// Mitsubishi GX Works2 project: exam_prep_diagrams   PLC: Q02/Q02H

PROGRAM complex1
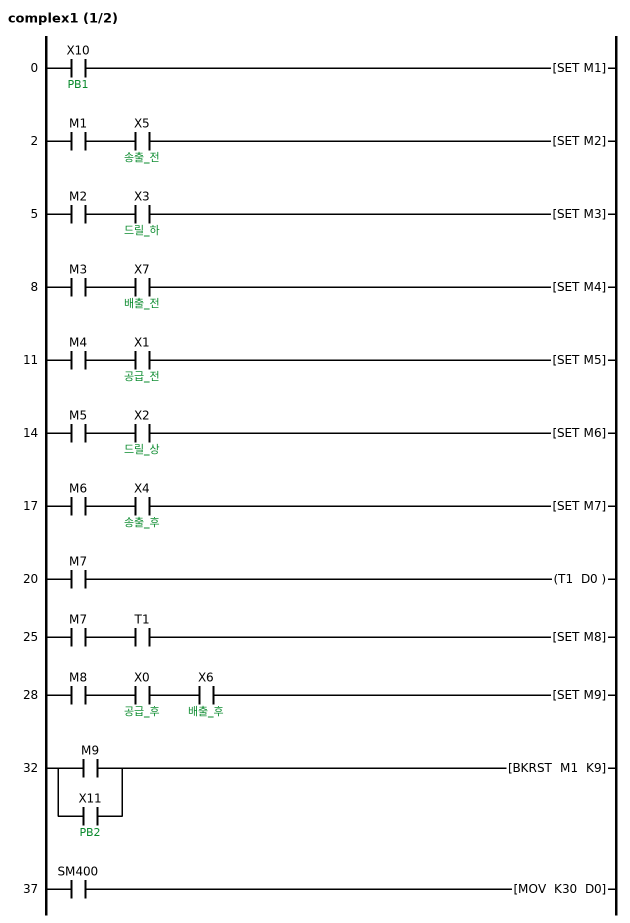
0     LD      X10  ; PB1
      SET     M1
2     LD      M1
      AND     X5  ; 송출_전
      SET     M2
5     LD      M2
      AND     X3  ; 드릴_하
      SET     M3
8     LD      M3
      AND     X7  ; 배출_전
      SET     M4
11    LD      M4
      AND     X1  ; 공급_전
      SET     M5
14    LD      M5
      AND     X2  ; 드릴_상
      SET     M6
17    LD      M6
      AND     X4  ; 송출_후
      SET     M7
20    LD      M7
      OUT     T1 D0
25    LD      M7
      AND     T1
      SET     M8
28    LD      M8
      AND     X0  ; 공급_후
      AND     X6  ; 배출_후
      SET     M9
32    LD      M9
      OR      X11  ; PB2
      BKRST   M1 K9
37    LD      SM400
      MOV     K30 D0
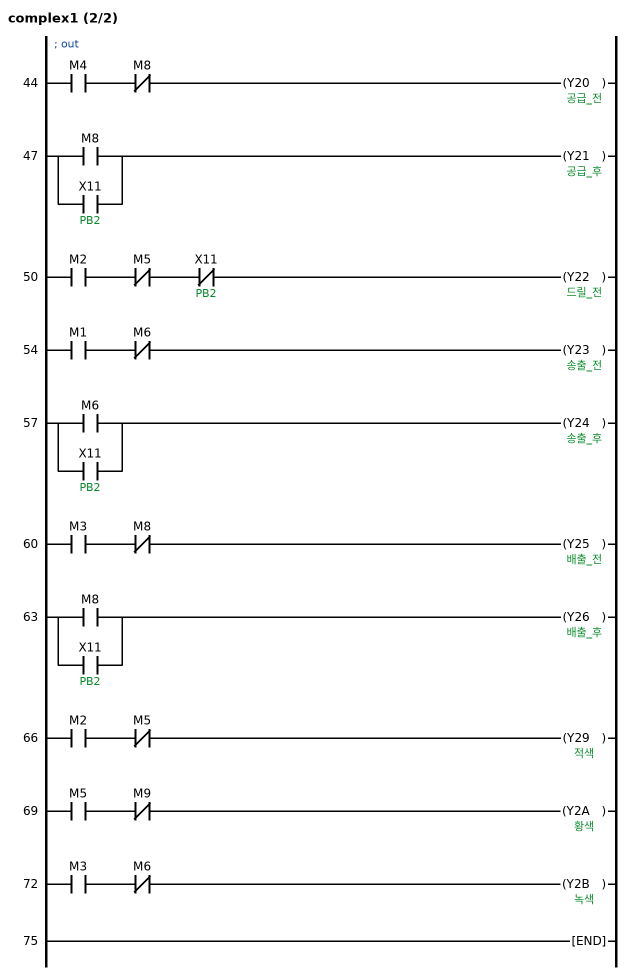
; out
44    LD      M4
      ANI     M8
      OUT     Y20  ; 공급_전
47    LD      M8
      OR      X11  ; PB2
      OUT     Y21  ; 공급_후
50    LD      M2
      ANI     M5
      ANI     X11  ; PB2
      OUT     Y22  ; 드릴_전
54    LD      M1
      ANI     M6
      OUT     Y23  ; 송출_전
57    LD      M6
      OR      X11  ; PB2
      OUT     Y24  ; 송출_후
60    LD      M3
      ANI     M8
      OUT     Y25  ; 배출_전
63    LD      M8
      OR      X11  ; PB2
      OUT     Y26  ; 배출_후
66    LD      M2
      ANI     M5
      OUT     Y29  ; 적색
69    LD      M5
      ANI     M9
      OUT     Y2A  ; 황색
72    LD      M3
      ANI     M6
      OUT     Y2B  ; 녹색
75    END
END_PROGRAM

PROGRAM complex2
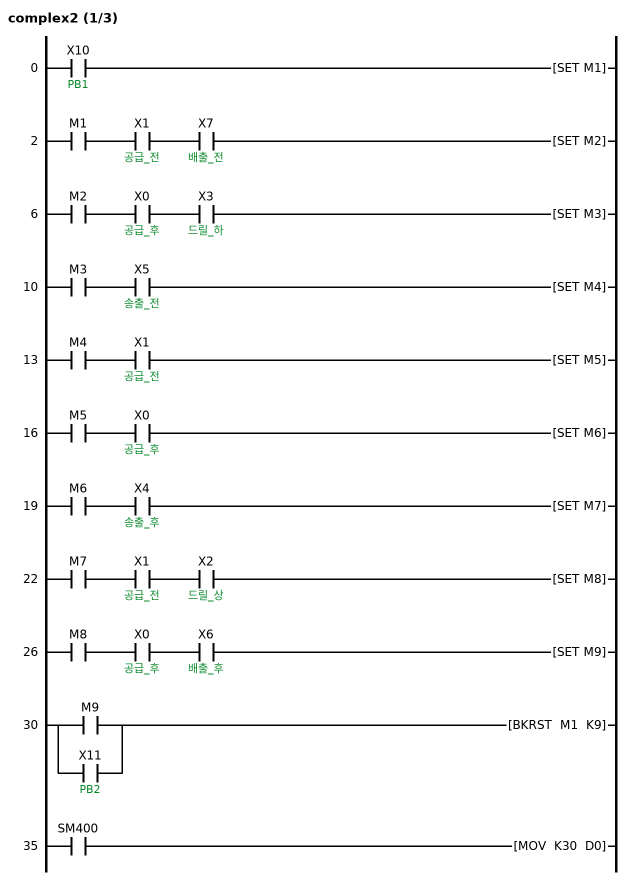
0     LD      X10  ; PB1
      SET     M1
2     LD      M1
      AND     X1  ; 공급_전
      AND     X7  ; 배출_전
      SET     M2
6     LD      M2
      AND     X0  ; 공급_후
      AND     X3  ; 드릴_하
      SET     M3
10    LD      M3
      AND     X5  ; 송출_전
      SET     M4
13    LD      M4
      AND     X1  ; 공급_전
      SET     M5
16    LD      M5
      AND     X0  ; 공급_후
      SET     M6
19    LD      M6
      AND     X4  ; 송출_후
      SET     M7
22    LD      M7
      AND     X1  ; 공급_전
      AND     X2  ; 드릴_상
      SET     M8
26    LD      M8
      AND     X0  ; 공급_후
      AND     X6  ; 배출_후
      SET     M9
30    LD      M9
      OR      X11  ; PB2
      BKRST   M1 K9
35    LD      SM400
      MOV     K30 D0
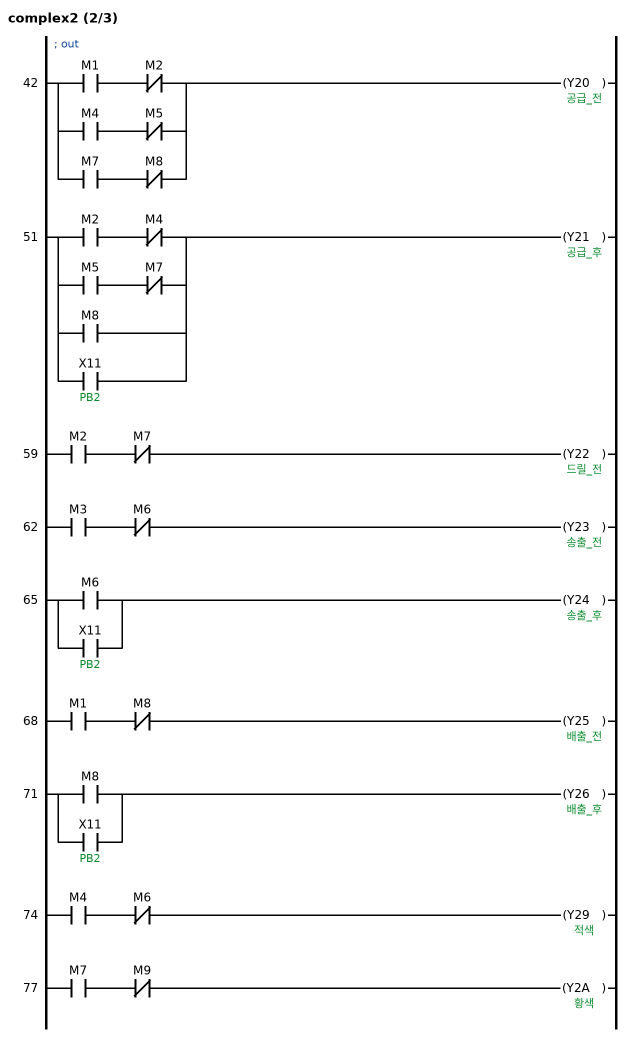
; out
42    LD      M1
      ANI     M2
      LD      M4
      ANI     M5
      ORB
      LD      M7
      ANI     M8
      ORB
      OUT     Y20  ; 공급_전
51    LD      M2
      ANI     M4
      LD      M5
      ANI     M7
      ORB
      OR      M8
      OR      X11  ; PB2
      OUT     Y21  ; 공급_후
59    LD      M2
      ANI     M7
      OUT     Y22  ; 드릴_전
62    LD      M3
      ANI     M6
      OUT     Y23  ; 송출_전
65    LD      M6
      OR      X11  ; PB2
      OUT     Y24  ; 송출_후
68    LD      M1
      ANI     M8
      OUT     Y25  ; 배출_전
71    LD      M8
      OR      X11  ; PB2
      OUT     Y26  ; 배출_후
74    LD      M4
      ANI     M6
      OUT     Y29  ; 적색
77    LD      M7
      ANI     M9
      OUT     Y2A  ; 황색
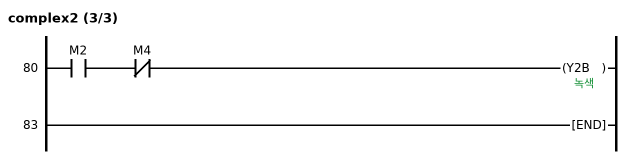
80    LD      M2
      ANI     M4
      OUT     Y2B  ; 녹색
83    END
END_PROGRAM

PROGRAM base
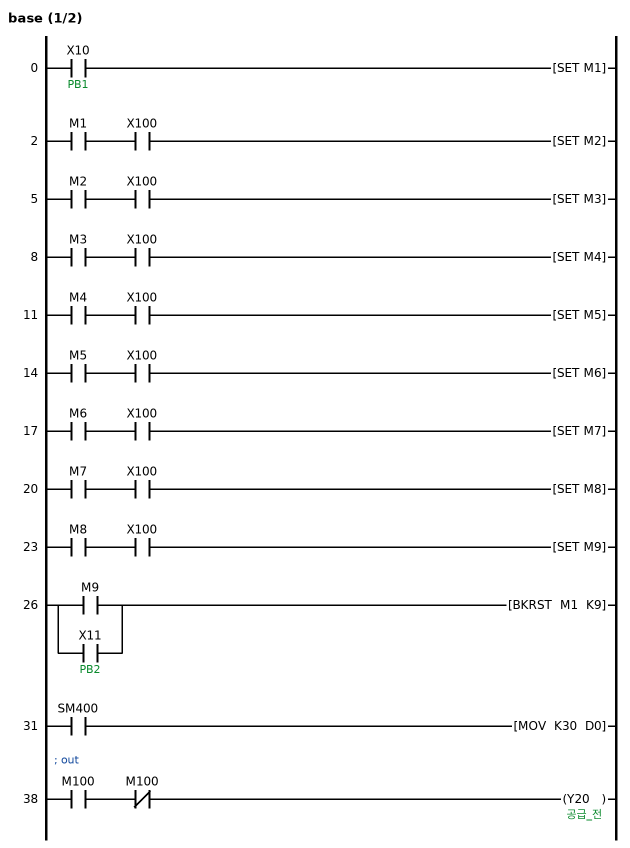
0     LD      X10  ; PB1
      SET     M1
2     LD      M1
      AND     X100
      SET     M2
5     LD      M2
      AND     X100
      SET     M3
8     LD      M3
      AND     X100
      SET     M4
11    LD      M4
      AND     X100
      SET     M5
14    LD      M5
      AND     X100
      SET     M6
17    LD      M6
      AND     X100
      SET     M7
20    LD      M7
      AND     X100
      SET     M8
23    LD      M8
      AND     X100
      SET     M9
26    LD      M9
      OR      X11  ; PB2
      BKRST   M1 K9
31    LD      SM400
      MOV     K30 D0
; out
38    LD      M100
      ANI     M100
      OUT     Y20  ; 공급_전
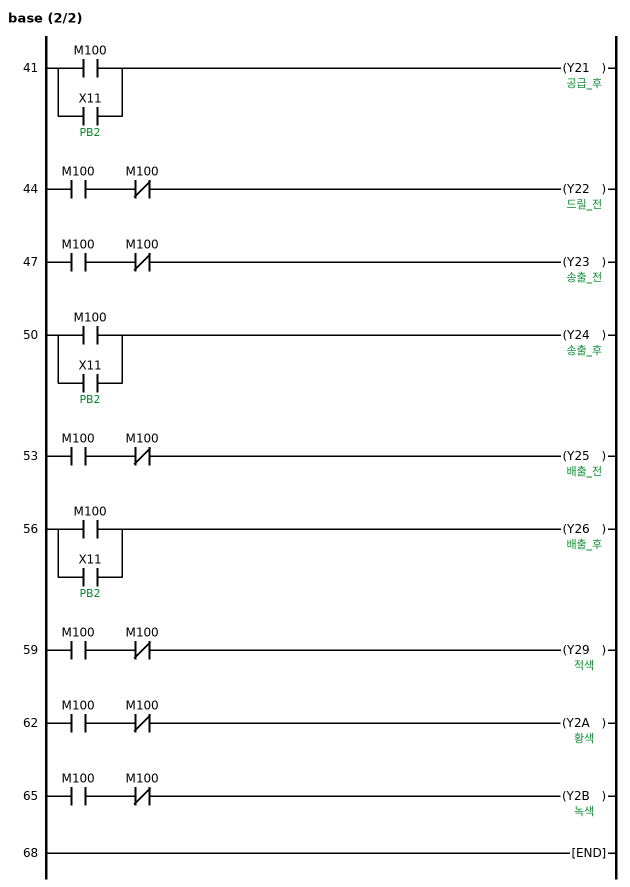
41    LD      M100
      OR      X11  ; PB2
      OUT     Y21  ; 공급_후
44    LD      M100
      ANI     M100
      OUT     Y22  ; 드릴_전
47    LD      M100
      ANI     M100
      OUT     Y23  ; 송출_전
50    LD      M100
      OR      X11  ; PB2
      OUT     Y24  ; 송출_후
53    LD      M100
      ANI     M100
      OUT     Y25  ; 배출_전
56    LD      M100
      OR      X11  ; PB2
      OUT     Y26  ; 배출_후
59    LD      M100
      ANI     M100
      OUT     Y29  ; 적색
62    LD      M100
      ANI     M100
      OUT     Y2A  ; 황색
65    LD      M100
      ANI     M100
      OUT     Y2B  ; 녹색
68    END
END_PROGRAM

PROGRAM complex3
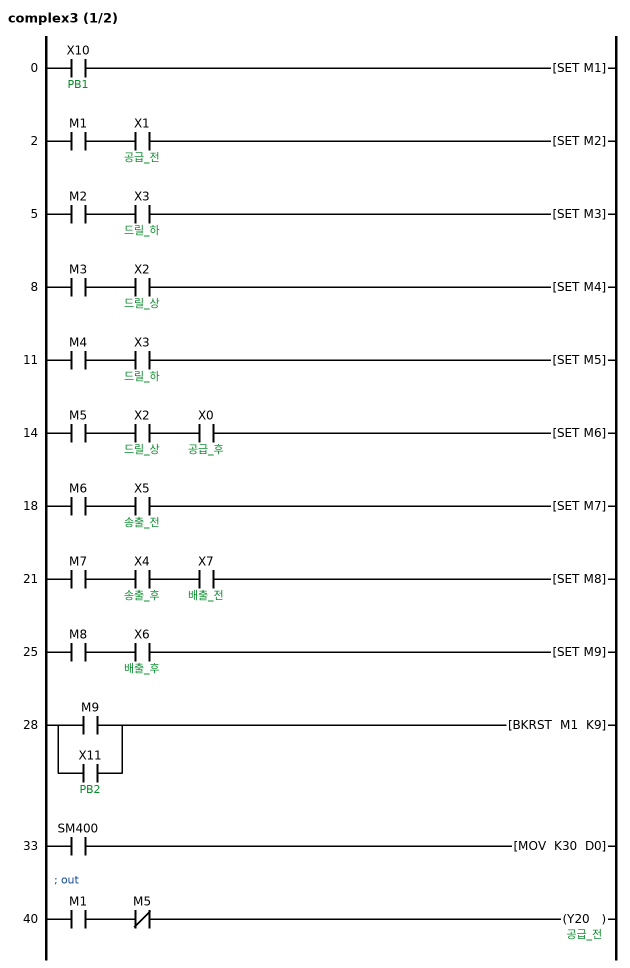
0     LD      X10  ; PB1
      SET     M1
2     LD      M1
      AND     X1  ; 공급_전
      SET     M2
5     LD      M2
      AND     X3  ; 드릴_하
      SET     M3
8     LD      M3
      AND     X2  ; 드릴_상
      SET     M4
11    LD      M4
      AND     X3  ; 드릴_하
      SET     M5
14    LD      M5
      AND     X2  ; 드릴_상
      AND     X0  ; 공급_후
      SET     M6
18    LD      M6
      AND     X5  ; 송출_전
      SET     M7
21    LD      M7
      AND     X4  ; 송출_후
      AND     X7  ; 배출_전
      SET     M8
25    LD      M8
      AND     X6  ; 배출_후
      SET     M9
28    LD      M9
      OR      X11  ; PB2
      BKRST   M1 K9
33    LD      SM400
      MOV     K30 D0
; out
40    LD      M1
      ANI     M5
      OUT     Y20  ; 공급_전
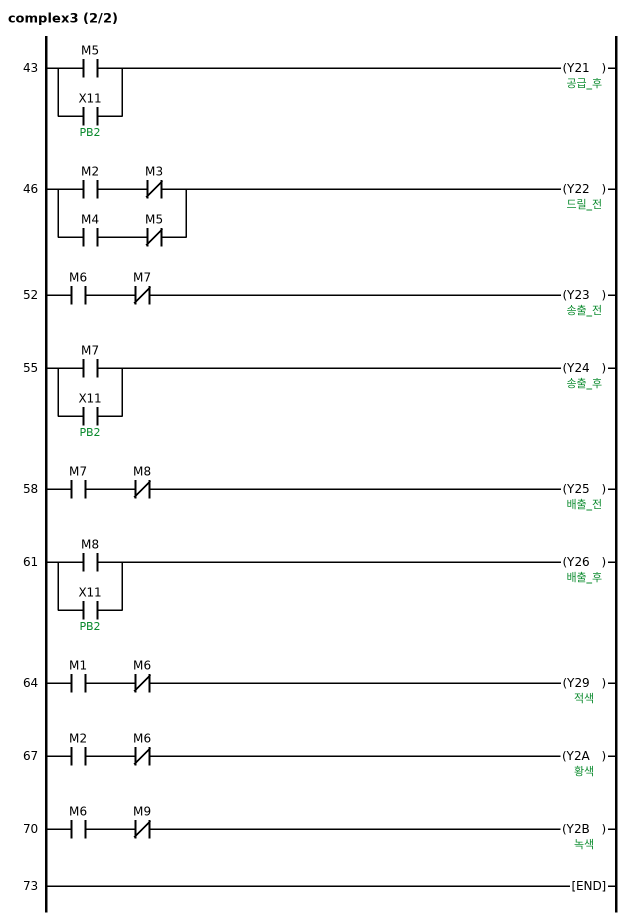
43    LD      M5
      OR      X11  ; PB2
      OUT     Y21  ; 공급_후
46    LD      M2
      ANI     M3
      LD      M4
      ANI     M5
      ORB
      OUT     Y22  ; 드릴_전
52    LD      M6
      ANI     M7
      OUT     Y23  ; 송출_전
55    LD      M7
      OR      X11  ; PB2
      OUT     Y24  ; 송출_후
58    LD      M7
      ANI     M8
      OUT     Y25  ; 배출_전
61    LD      M8
      OR      X11  ; PB2
      OUT     Y26  ; 배출_후
64    LD      M1
      ANI     M6
      OUT     Y29  ; 적색
67    LD      M2
      ANI     M6
      OUT     Y2A  ; 황색
70    LD      M6
      ANI     M9
      OUT     Y2B  ; 녹색
73    END
END_PROGRAM

PROGRAM EXAM1
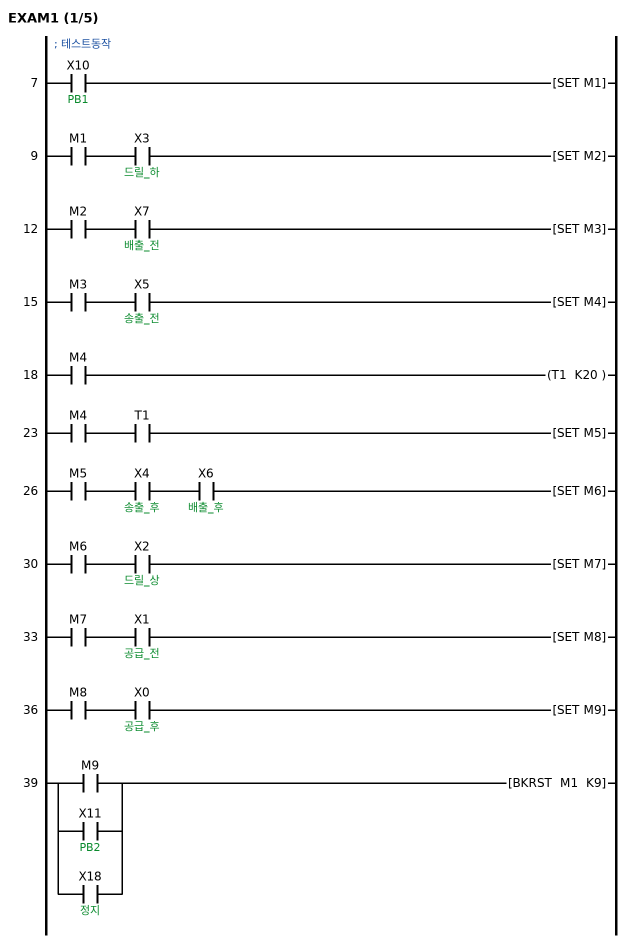
; 테스트동작
7     LD      X10  ; PB1
      SET     M1
9     LD      M1
      AND     X3  ; 드릴_하
      SET     M2
12    LD      M2
      AND     X7  ; 배출_전
      SET     M3
15    LD      M3
      AND     X5  ; 송출_전
      SET     M4
18    LD      M4
      OUT     T1 K20
23    LD      M4
      AND     T1
      SET     M5
26    LD      M5
      AND     X4  ; 송출_후
      AND     X6  ; 배출_후
      SET     M6
30    LD      M6
      AND     X2  ; 드릴_상
      SET     M7
33    LD      M7
      AND     X1  ; 공급_전
      SET     M8
36    LD      M8
      AND     X0  ; 공급_후
      SET     M9
39    LD      M9
      OR      X11  ; PB2
      OR      X18  ; 정지
      BKRST   M1 K9
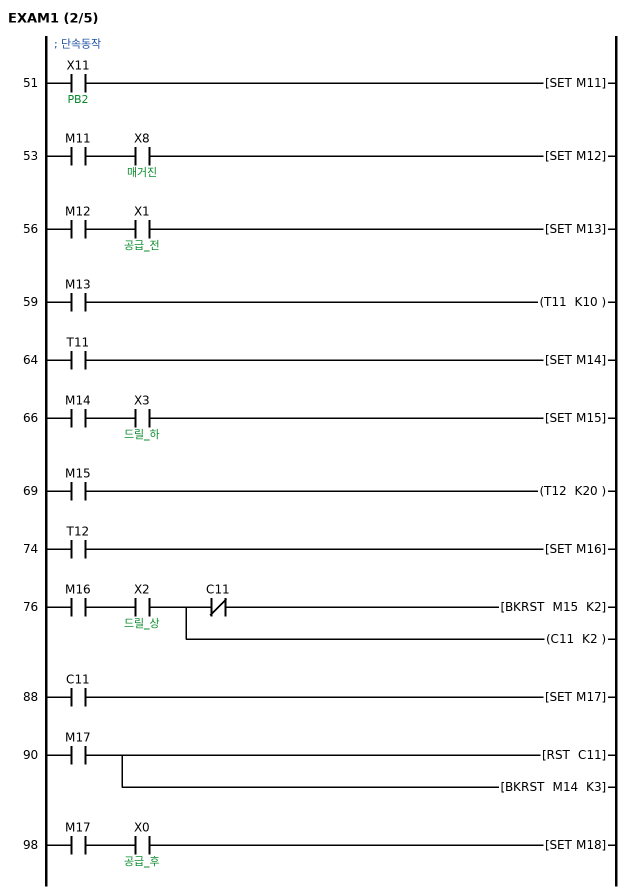
; 단속동작
51    LD      X11  ; PB2
      SET     M11
53    LD      M11
      AND     X8  ; 매거진
      SET     M12
56    LD      M12
      AND     X1  ; 공급_전
      SET     M13
59    LD      M13
      OUT     T11 K10
64    LD      T11
      SET     M14
66    LD      M14
      AND     X3  ; 드릴_하
      SET     M15
69    LD      M15
      OUT     T12 K20
74    LD      T12
      SET     M16
76    LD      M16
      AND     X2  ; 드릴_상
      MPS
      ANI     C11
      BKRST   M15 K2
      MPP
      OUT     C11 K2
88    LD      C11
      SET     M17
90    LD      M17
      RST     C11
      BKRST   M14 K3
98    LD      M17
      AND     X0  ; 공급_후
      SET     M18
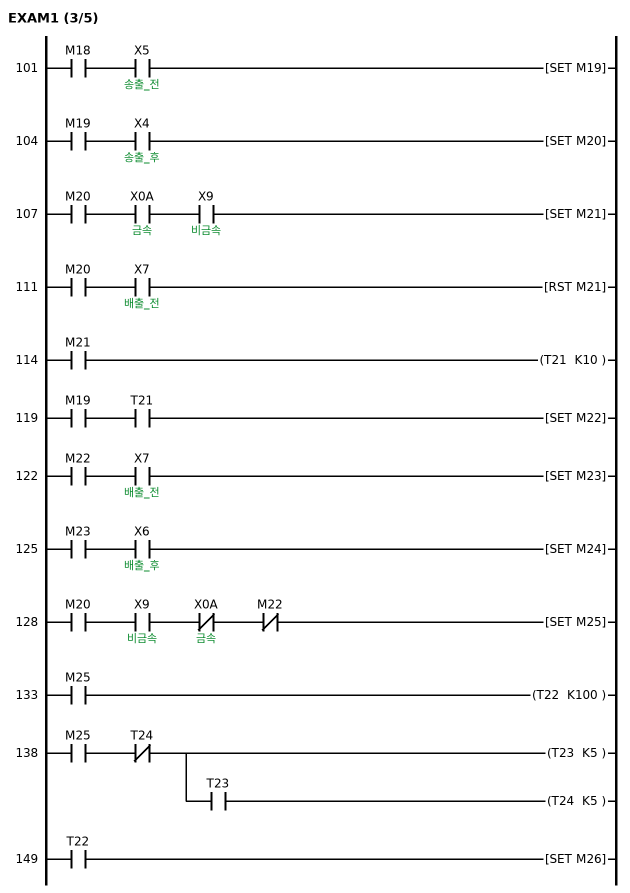
101   LD      M18
      AND     X5  ; 송출_전
      SET     M19
104   LD      M19
      AND     X4  ; 송출_후
      SET     M20
107   LD      M20
      AND     X0A  ; 금속
      AND     X9  ; 비금속
      SET     M21
111   LD      M20
      AND     X7  ; 배출_전
      RST     M21
114   LD      M21
      OUT     T21 K10
119   LD      M19
      AND     T21
      SET     M22
122   LD      M22
      AND     X7  ; 배출_전
      SET     M23
125   LD      M23
      AND     X6  ; 배출_후
      SET     M24
128   LD      M20
      AND     X9  ; 비금속
      ANI     X0A  ; 금속
      ANI     M22
      SET     M25
133   LD      M25
      OUT     T22 K100
138   LD      M25
      ANI     T24
      OUT     T23 K5
      AND     T23
      OUT     T24 K5
149   LD      T22
      SET     M26
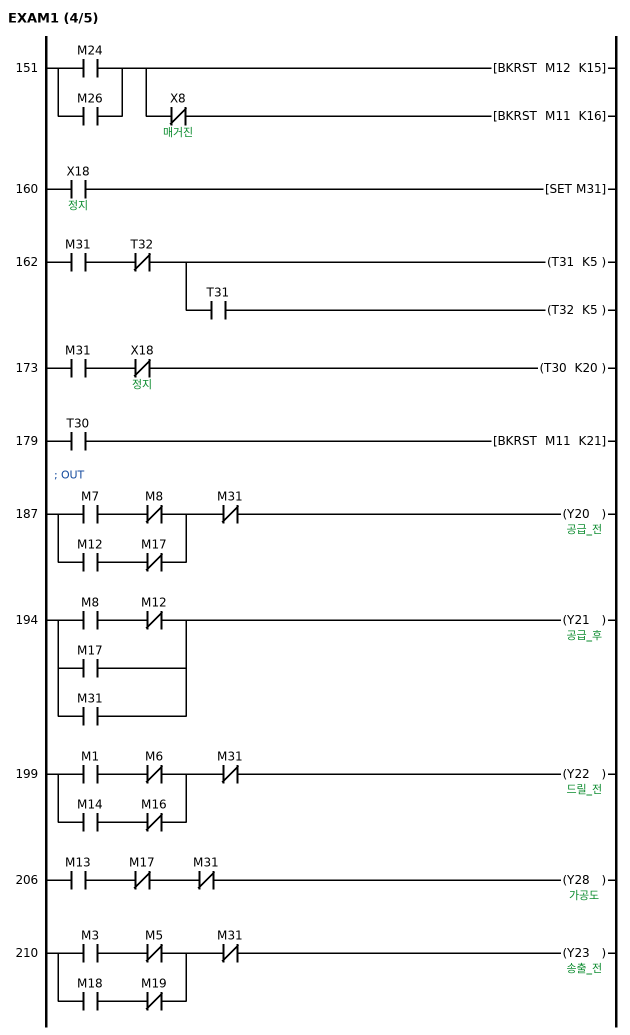
151   LD      M24
      OR      M26
      BKRST   M12 K15
      ANI     X8  ; 매거진
      BKRST   M11 K16
160   LD      X18  ; 정지
      SET     M31
162   LD      M31
      ANI     T32
      OUT     T31 K5
      AND     T31
      OUT     T32 K5
173   LD      M31
      ANI     X18  ; 정지
      OUT     T30 K20
179   LD      T30
      BKRST   M11 K21
; OUT
187   LD      M7
      ANI     M8
      LD      M12
      ANI     M17
      ORB
      ANI     M31
      OUT     Y20  ; 공급_전
194   LD      M8
      ANI     M12
      OR      M17
      OR      M31
      OUT     Y21  ; 공급_후
199   LD      M1
      ANI     M6
      LD      M14
      ANI     M16
      ORB
      ANI     M31
      OUT     Y22  ; 드릴_전
206   LD      M13
      ANI     M17
      ANI     M31
      OUT     Y28  ; 가공도
210   LD      M3
      ANI     M5
      LD      M18
      ANI     M19
      ORB
      ANI     M31
      OUT     Y23  ; 송출_전
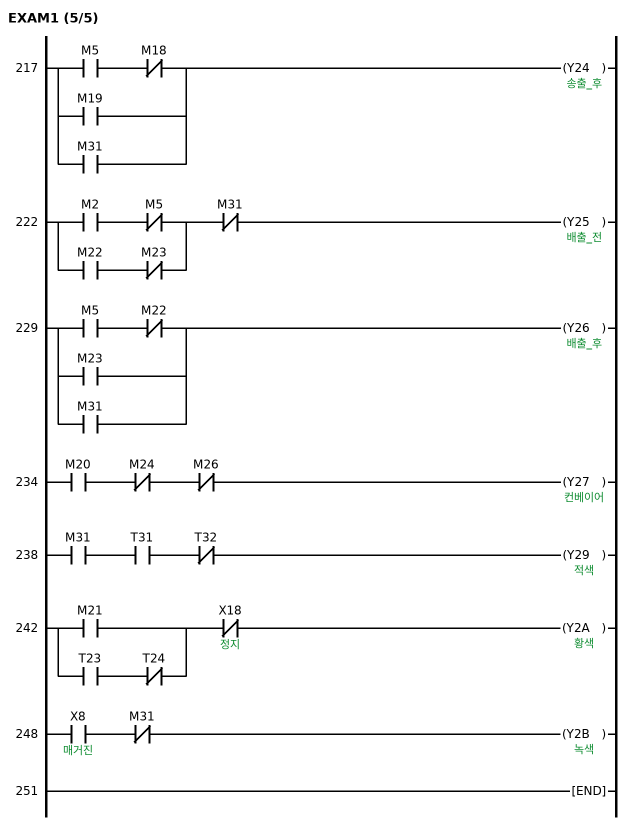
217   LD      M5
      ANI     M18
      OR      M19
      OR      M31
      OUT     Y24  ; 송출_후
222   LD      M2
      ANI     M5
      LD      M22
      ANI     M23
      ORB
      ANI     M31
      OUT     Y25  ; 배출_전
229   LD      M5
      ANI     M22
      OR      M23
      OR      M31
      OUT     Y26  ; 배출_후
234   LD      M20
      ANI     M24
      ANI     M26
      OUT     Y27  ; 컨베이어
238   LD      M31
      AND     T31
      ANI     T32
      OUT     Y29  ; 적색
242   LD      M21
      LD      T23
      ANI     T24
      ORB
      ANI     X18  ; 정지
      OUT     Y2A  ; 황색
248   LD      X8  ; 매거진
      ANI     M31
      OUT     Y2B  ; 녹색
251   END
END_PROGRAM

PROGRAM practice
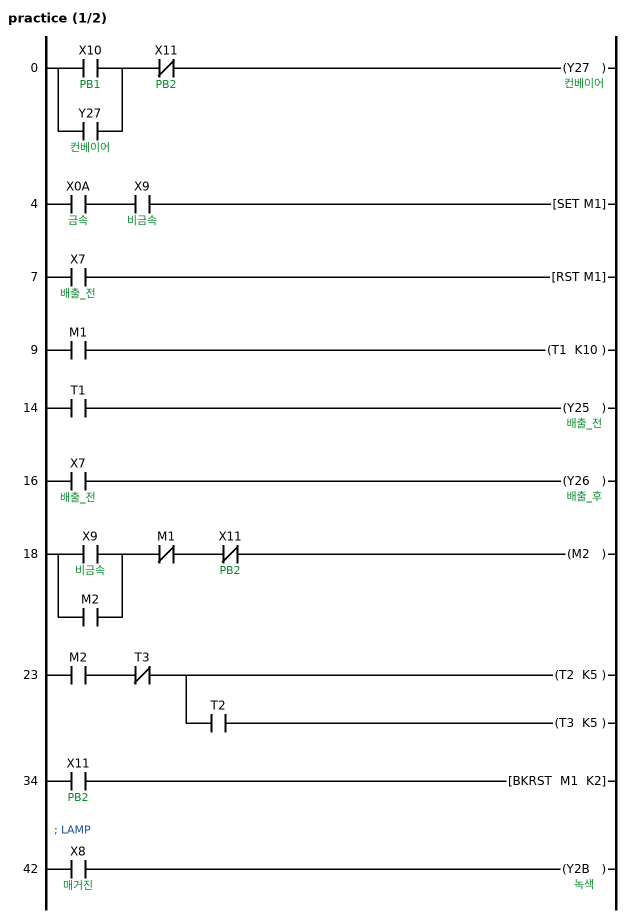
0     LD      X10  ; PB1
      OR      Y27  ; 컨베이어
      ANI     X11  ; PB2
      OUT     Y27  ; 컨베이어
4     LD      X0A  ; 금속
      AND     X9  ; 비금속
      SET     M1
7     LD      X7  ; 배출_전
      RST     M1
9     LD      M1
      OUT     T1 K10
14    LD      T1
      OUT     Y25  ; 배출_전
16    LD      X7  ; 배출_전
      OUT     Y26  ; 배출_후
18    LD      X9  ; 비금속
      OR      M2
      ANI     M1
      ANI     X11  ; PB2
      OUT     M2
23    LD      M2
      ANI     T3
      OUT     T2 K5
      AND     T2
      OUT     T3 K5
34    LD      X11  ; PB2
      BKRST   M1 K2
; LAMP
42    LD      X8  ; 매거진
      OUT     Y2B  ; 녹색
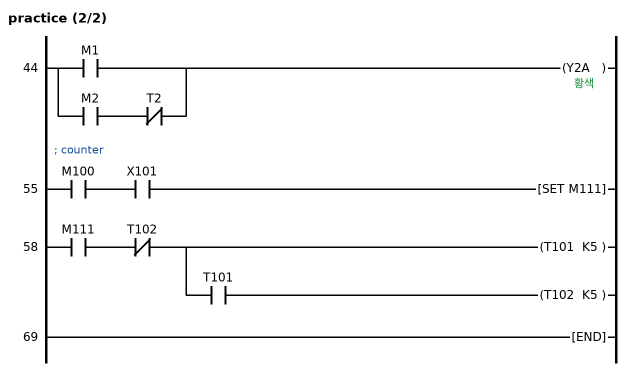
44    LD      M1
      LD      M2
      ANI     T2
      ORB
      OUT     Y2A  ; 황색
; counter
55    LD      M100
      AND     X101
      SET     M111
58    LD      M111
      ANI     T102
      OUT     T101 K5
      AND     T101
      OUT     T102 K5
69    END
END_PROGRAM

PROGRAM EXAM2
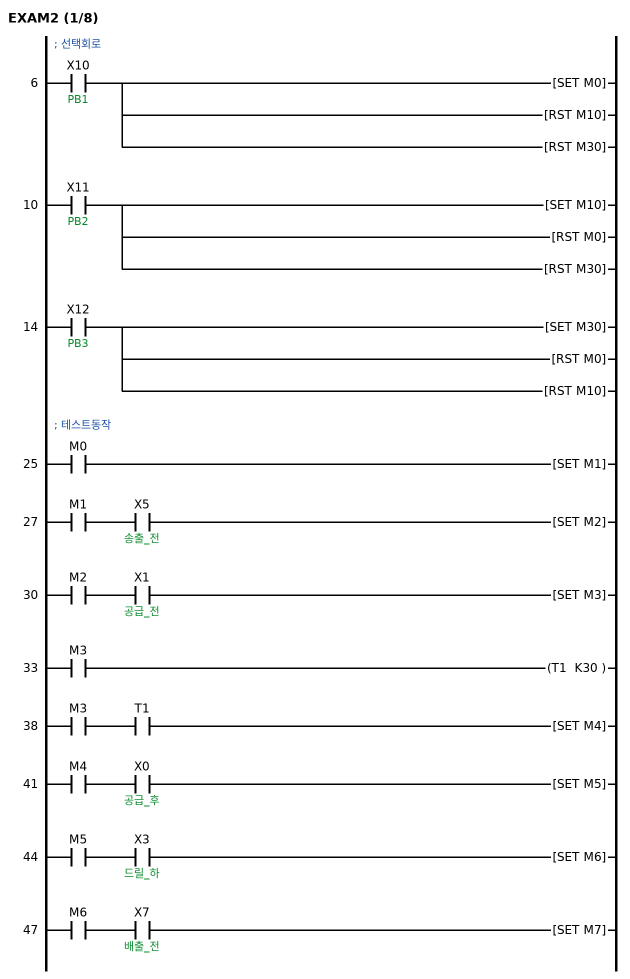
; 선택회로
6     LD      X10  ; PB1
      SET     M0
      RST     M10
      RST     M30
10    LD      X11  ; PB2
      SET     M10
      RST     M0
      RST     M30
14    LD      X12  ; PB3
      SET     M30
      RST     M0
      RST     M10
; 테스트동작
25    LD      M0
      SET     M1
27    LD      M1
      AND     X5  ; 송출_전
      SET     M2
30    LD      M2
      AND     X1  ; 공급_전
      SET     M3
33    LD      M3
      OUT     T1 K30
38    LD      M3
      AND     T1
      SET     M4
41    LD      M4
      AND     X0  ; 공급_후
      SET     M5
44    LD      M5
      AND     X3  ; 드릴_하
      SET     M6
47    LD      M6
      AND     X7  ; 배출_전
      SET     M7
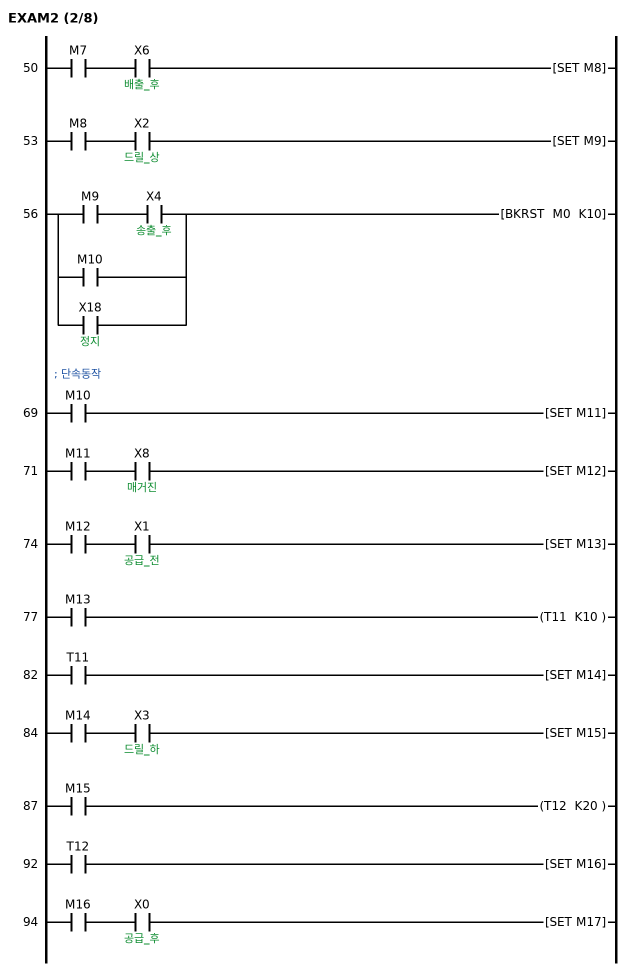
50    LD      M7
      AND     X6  ; 배출_후
      SET     M8
53    LD      M8
      AND     X2  ; 드릴_상
      SET     M9
56    LD      M9
      AND     X4  ; 송출_후
      OR      M10
      OR      X18  ; 정지
      BKRST   M0 K10
; 단속동작
69    LD      M10
      SET     M11
71    LD      M11
      AND     X8  ; 매거진
      SET     M12
74    LD      M12
      AND     X1  ; 공급_전
      SET     M13
77    LD      M13
      OUT     T11 K10
82    LD      T11
      SET     M14
84    LD      M14
      AND     X3  ; 드릴_하
      SET     M15
87    LD      M15
      OUT     T12 K20
92    LD      T12
      SET     M16
94    LD      M16
      AND     X0  ; 공급_후
      SET     M17
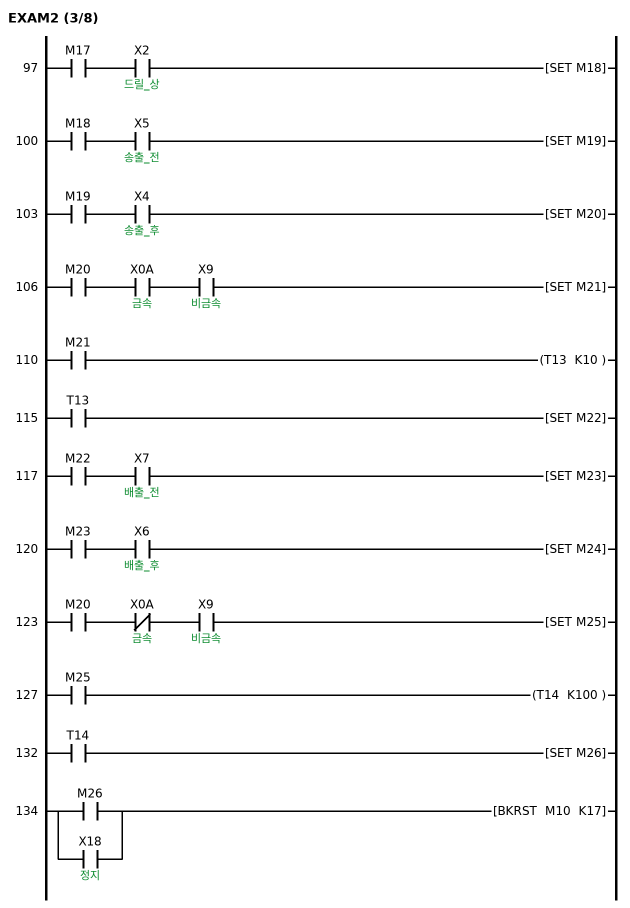
97    LD      M17
      AND     X2  ; 드릴_상
      SET     M18
100   LD      M18
      AND     X5  ; 송출_전
      SET     M19
103   LD      M19
      AND     X4  ; 송출_후
      SET     M20
106   LD      M20
      AND     X0A  ; 금속
      AND     X9  ; 비금속
      SET     M21
110   LD      M21
      OUT     T13 K10
115   LD      T13
      SET     M22
117   LD      M22
      AND     X7  ; 배출_전
      SET     M23
120   LD      M23
      AND     X6  ; 배출_후
      SET     M24
123   LD      M20
      ANI     X0A  ; 금속
      AND     X9  ; 비금속
      SET     M25
127   LD      M25
      OUT     T14 K100
132   LD      T14
      SET     M26
134   LD      M26
      OR      X18  ; 정지
      BKRST   M10 K17
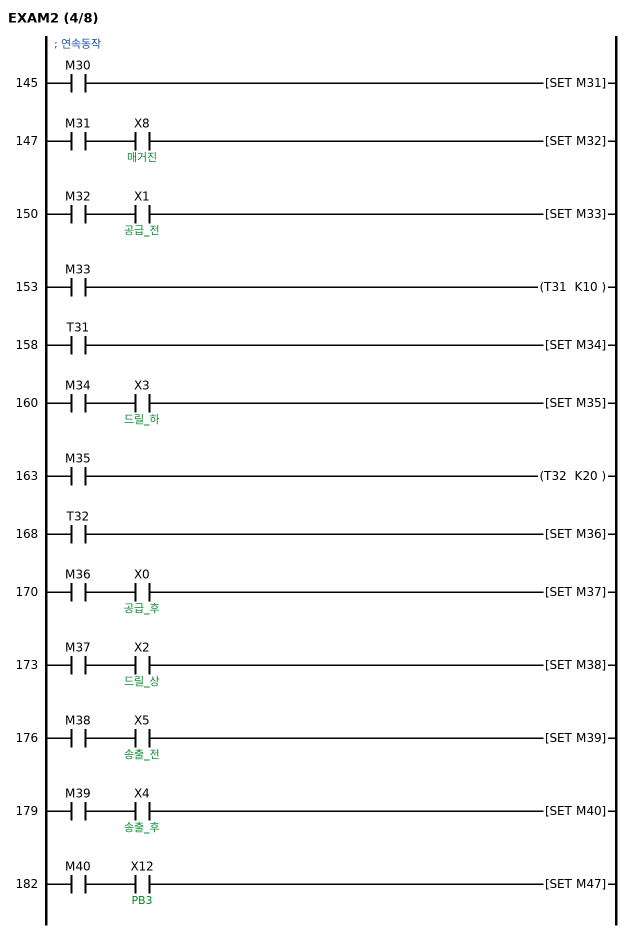
; 연속동작
145   LD      M30
      SET     M31
147   LD      M31
      AND     X8  ; 매거진
      SET     M32
150   LD      M32
      AND     X1  ; 공급_전
      SET     M33
153   LD      M33
      OUT     T31 K10
158   LD      T31
      SET     M34
160   LD      M34
      AND     X3  ; 드릴_하
      SET     M35
163   LD      M35
      OUT     T32 K20
168   LD      T32
      SET     M36
170   LD      M36
      AND     X0  ; 공급_후
      SET     M37
173   LD      M37
      AND     X2  ; 드릴_상
      SET     M38
176   LD      M38
      AND     X5  ; 송출_전
      SET     M39
179   LD      M39
      AND     X4  ; 송출_후
      SET     M40
182   LD      M40
      AND     X12  ; PB3
      SET     M47
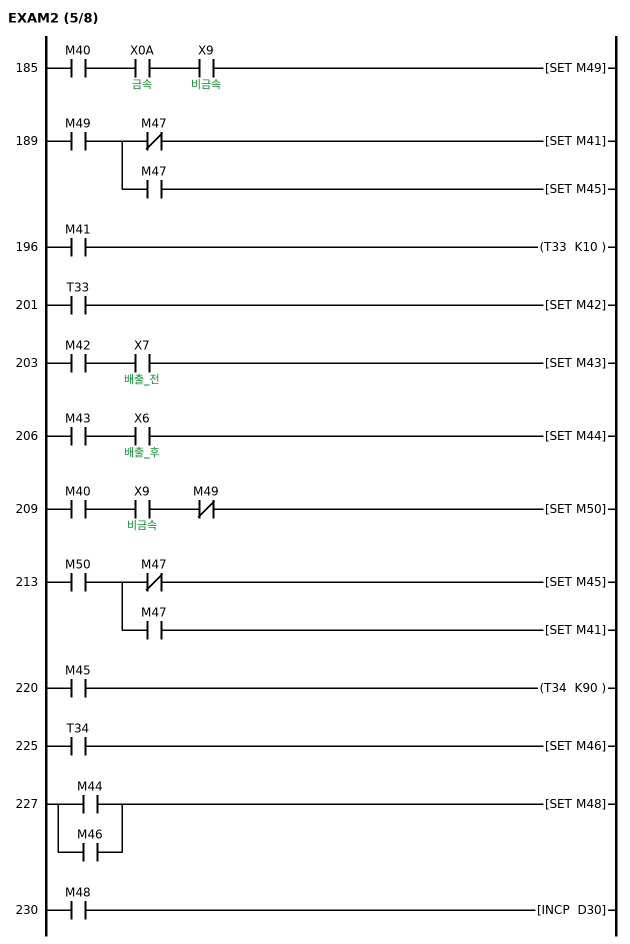
185   LD      M40
      AND     X0A  ; 금속
      AND     X9  ; 비금속
      SET     M49
189   LD      M49
      MPS
      ANI     M47
      SET     M41
      MPP
      AND     M47
      SET     M45
196   LD      M41
      OUT     T33 K10
201   LD      T33
      SET     M42
203   LD      M42
      AND     X7  ; 배출_전
      SET     M43
206   LD      M43
      AND     X6  ; 배출_후
      SET     M44
209   LD      M40
      AND     X9  ; 비금속
      ANI     M49
      SET     M50
213   LD      M50
      MPS
      ANI     M47
      SET     M45
      MPP
      AND     M47
      SET     M41
220   LD      M45
      OUT     T34 K90
225   LD      T34
      SET     M46
227   LD      M44
      OR      M46
      SET     M48
230   LD      M48
      INCP    D30
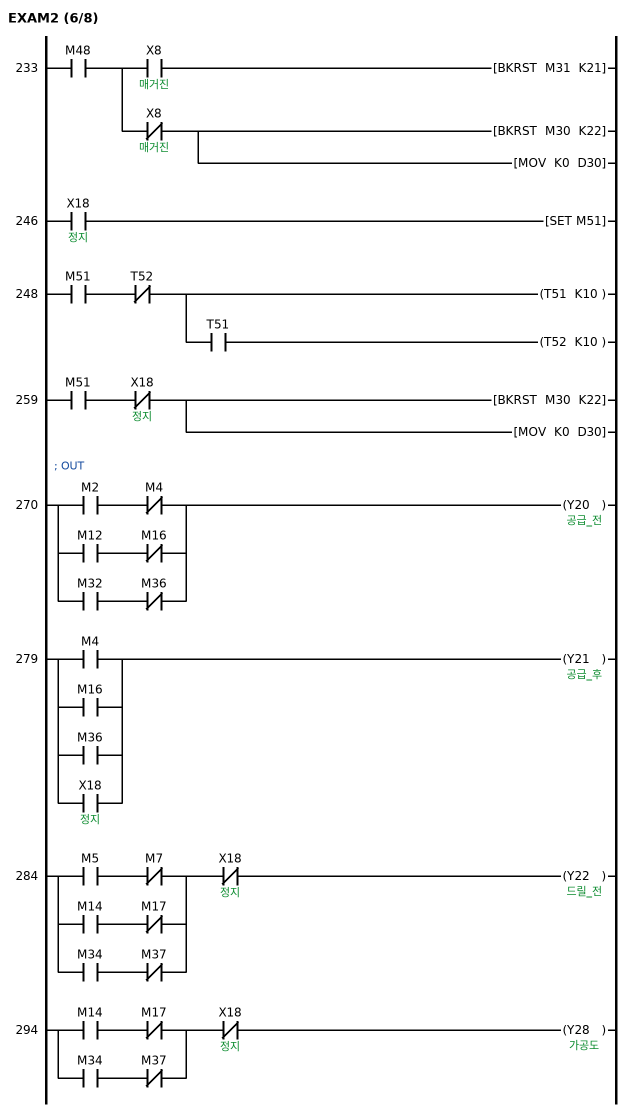
233   LD      M48
      MPS
      AND     X8  ; 매거진
      BKRST   M31 K21
      MPP
      ANI     X8  ; 매거진
      BKRST   M30 K22
      MOV     K0 D30
246   LD      X18  ; 정지
      SET     M51
248   LD      M51
      ANI     T52
      OUT     T51 K10
      AND     T51
      OUT     T52 K10
259   LD      M51
      ANI     X18  ; 정지
      BKRST   M30 K22
      MOV     K0 D30
; OUT
270   LD      M2
      ANI     M4
      LD      M12
      ANI     M16
      ORB
      LD      M32
      ANI     M36
      ORB
      OUT     Y20  ; 공급_전
279   LD      M4
      OR      M16
      OR      M36
      OR      X18  ; 정지
      OUT     Y21  ; 공급_후
284   LD      M5
      ANI     M7
      LD      M14
      ANI     M17
      ORB
      LD      M34
      ANI     M37
      ORB
      ANI     X18  ; 정지
      OUT     Y22  ; 드릴_전
294   LD      M14
      ANI     M17
      LD      M34
      ANI     M37
      ORB
      ANI     X18  ; 정지
      OUT     Y28  ; 가공도
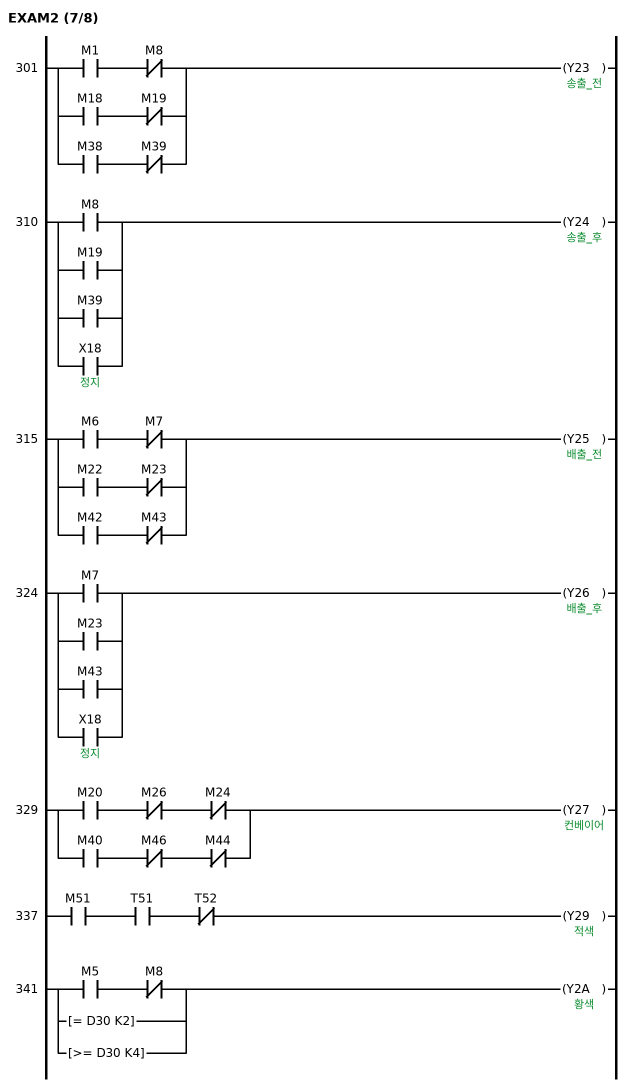
301   LD      M1
      ANI     M8
      LD      M18
      ANI     M19
      ORB
      LD      M38
      ANI     M39
      ORB
      OUT     Y23  ; 송출_전
310   LD      M8
      OR      M19
      OR      M39
      OR      X18  ; 정지
      OUT     Y24  ; 송출_후
315   LD      M6
      ANI     M7
      LD      M22
      ANI     M23
      ORB
      LD      M42
      ANI     M43
      ORB
      OUT     Y25  ; 배출_전
324   LD      M7
      OR      M23
      OR      M43
      OR      X18  ; 정지
      OUT     Y26  ; 배출_후
329   LD      M20
      ANI     M26
      ANI     M24
      LD      M40
      ANI     M46
      ANI     M44
      ORB
      OUT     Y27  ; 컨베이어
337   LD      M51
      AND     T51
      ANI     T52
      OUT     Y29  ; 적색
341   LD      M5
      ANI     M8
      OR=     D30 K2
      OR>=    D30 K4
      OUT     Y2A  ; 황색
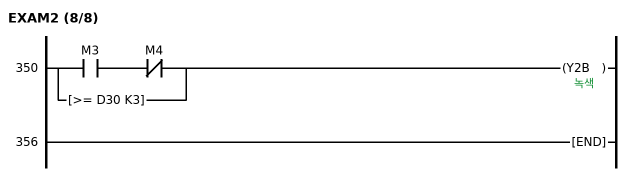
350   LD      M3
      ANI     M4
      OR>=    D30 K3
      OUT     Y2B  ; 녹색
356   END
END_PROGRAM

PROGRAM EXAM3
